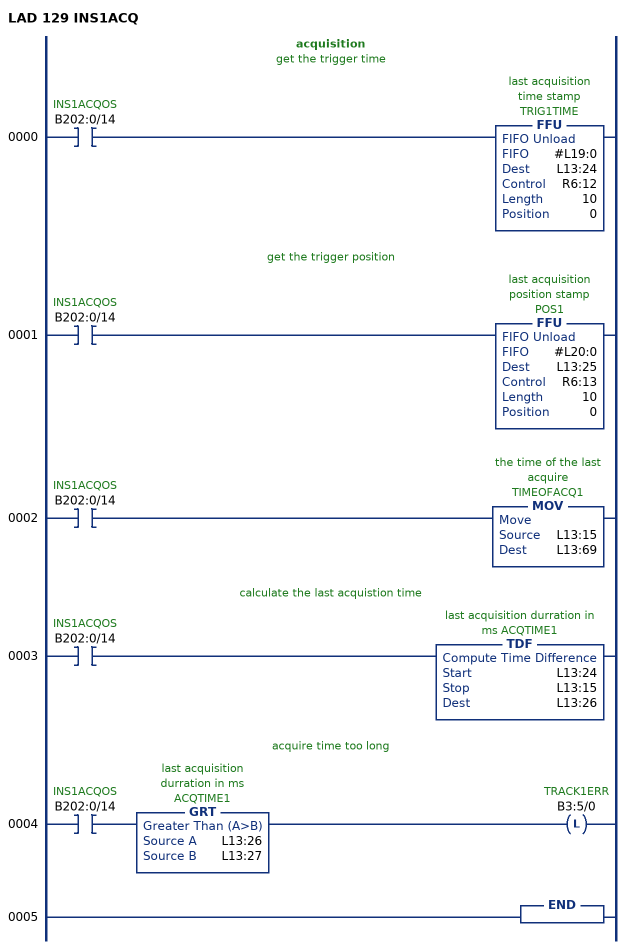
% Rung: 0 %
% TITLE: acquisition %
% get the trigger time %
SOR XIC B202:0/14 FFU #L19:0 L13:24 R6:12 10 0 EOR
%   B202:0/14  INS1ACQOS %
%   L13:24  TRIG1TIME  "last acquisition time stamp" %
% Rung: 1 %
% get the trigger position %
SOR XIC B202:0/14 FFU #L20:0 L13:25 R6:13 10 0 EOR
%   B202:0/14  INS1ACQOS %
%   L13:25  POS1  "last acquisition position stamp" %
% Rung: 2 %
SOR XIC B202:0/14 MOV L13:15 L13:69 EOR
%   B202:0/14  INS1ACQOS %
%   L13:15  THE_TIME %
%   L13:69  TIMEOFACQ1  "the time of the last acquire" %
% Rung: 3 %
% calculate the last acquistion time %
SOR XIC B202:0/14 TDF L13:24 L13:15 L13:26 EOR
%   B202:0/14  INS1ACQOS %
%   L13:24  TRIG1TIME  "last acquisition time stamp" %
%   L13:15  THE_TIME %
%   L13:26  ACQTIME1  "last acquisition durration in ms" %
% Rung: 4 %
% acquire time too long %
SOR XIC B202:0/14 GRT L13:26 L13:27 OTL B3:5/0 EOR
%   B202:0/14  INS1ACQOS %
%   L13:26  ACQTIME1  "last acquisition durration in ms" %
%   L13:27  "max acquisition time in ms" %
%   B3:5/0  TRACK1ERR %
% Rung: 5 %
SOR END EOR

LADDER 130 "INS1TRIG"
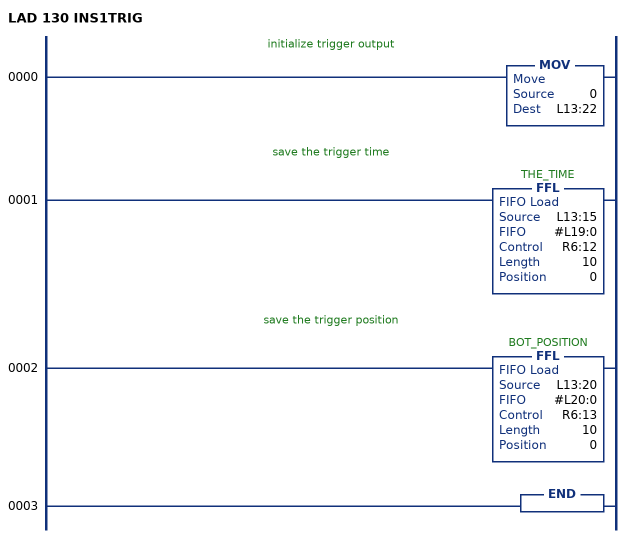
% Rung: 0 %
% initialize trigger output %
SOR MOV 0 L13:22 EOR
% Rung: 1 %
% save the trigger time %
SOR FFL L13:15 #L19:0 R6:12 10 0 EOR
%   L13:15  THE_TIME %
% Rung: 2 %
% save the trigger position %
SOR FFL L13:20 #L20:0 R6:13 10 0 EOR
%   L13:20  BOT_POSITION %
% Rung: 3 %
SOR END EOR

LADDER 131 "XFER"
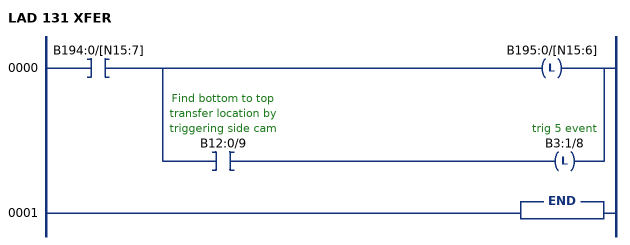
% Rung: 0 %
SOR XIC B194:0/[N15:7] BST OTL B195:0/[N15:6] NXB XIC B12:0/9 OTL B3:1/8 BND EOR
%   N15:7  XFER_OUT_LOC %
%   N15:6  XFER_IN_LOC %
%   B12:0/9  "Find bottom to top transfer location by triggering side cam" %
%   B3:1/8  "trig 5 event" %
% Rung: 1 %
SOR END EOR

LADDER 141 "OPTICTOP"
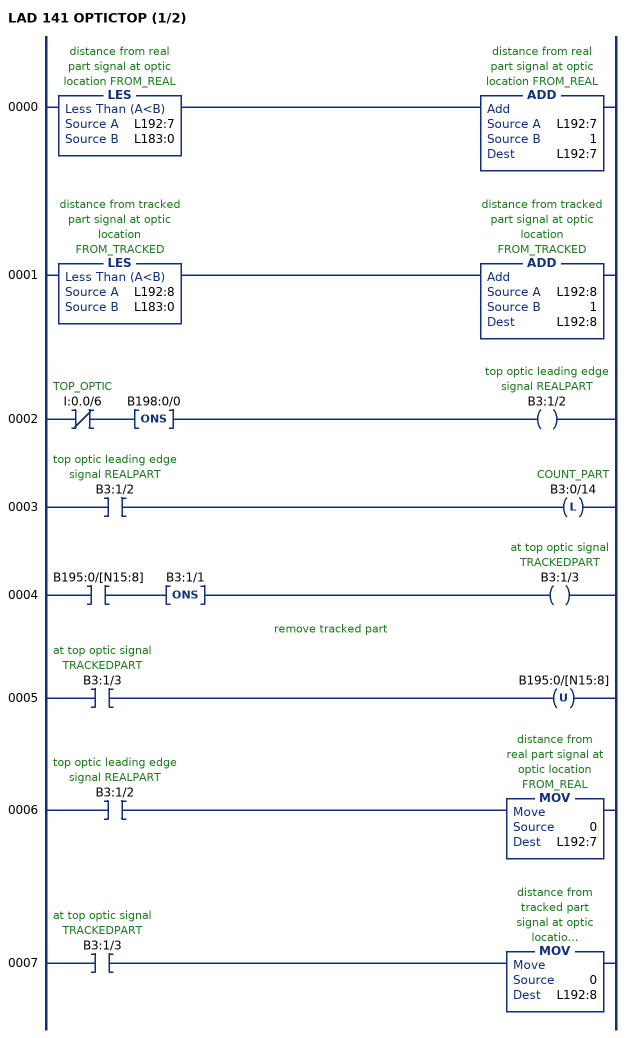
% Rung: 0 %
SOR LES L192:7 L183:0 ADD L192:7 1 L192:7 EOR
%   L192:7  FROM_REAL  "distance from real part signal at optic location" %
% Rung: 1 %
SOR LES L192:8 L183:0 ADD L192:8 1 L192:8 EOR
%   L192:8  FROM_TRACKED  "distance from tracked part signal at optic location" %
% Rung: 2 %
SOR XIO I:0.0/6 ONS B198:0/0 OTE B3:1/2 EOR
%   I:0.0/6  TOP_OPTIC %
%   B3:1/2  REALPART  "top optic leading edge signal" %
% Rung: 3 %
SOR XIC B3:1/2 OTL B3:0/14 EOR
%   B3:1/2  REALPART  "top optic leading edge signal" %
%   B3:0/14  COUNT_PART %
% Rung: 4 %
SOR XIC B195:0/[N15:8] ONS B3:1/1 OTE B3:1/3 EOR
%   N15:8  TOP_OPTIC_LOC %
%   B3:1/3  TRACKEDPART  "at top optic signal" %
% Rung: 5 %
% remove tracked part %
SOR XIC B3:1/3 OTU B195:0/[N15:8] EOR
%   B3:1/3  TRACKEDPART  "at top optic signal" %
%   N15:8  TOP_OPTIC_LOC %
% Rung: 6 %
SOR XIC B3:1/2 MOV 0 L192:7 EOR
%   B3:1/2  REALPART  "top optic leading edge signal" %
%   L192:7  FROM_REAL  "distance from real part signal at optic location" %
% Rung: 7 %
SOR XIC B3:1/3 MOV 0 L192:8 EOR
%   B3:1/3  TRACKEDPART  "at top optic signal" %
%   L192:8  FROM_TRACKED  "distance from tracked part signal at optic location" %

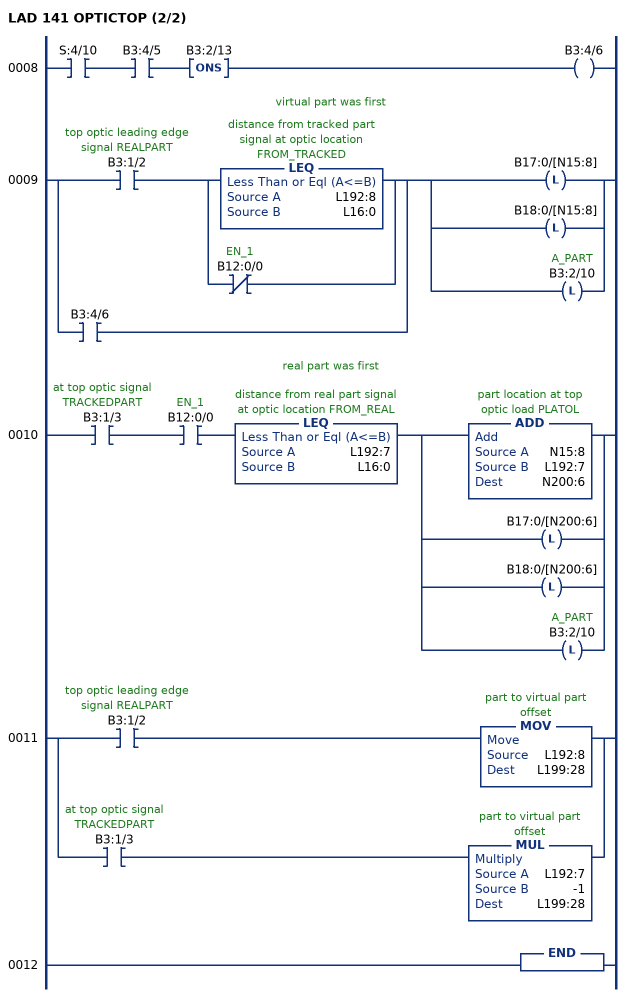
% Rung: 8 %
SOR XIC S:4/10 XIC B3:4/5 ONS B3:2/13 OTE B3:4/6 EOR
% Rung: 9 %
% virtual part was first %
SOR BST XIC B3:1/2 BST LEQ L192:8 L16:0 NXB XIO B12:0/0 BND NXB XIC B3:4/6 BND BST OTL B17:0/[N15:8] NXB OTL B18:0/[N15:8] NXB OTL B3:2/10 BND EOR
%   B3:1/2  REALPART  "top optic leading edge signal" %
%   L192:8  FROM_TRACKED  "distance from tracked part signal at optic location" %
%   B12:0/0  EN_1 %
%   N15:8  TOP_OPTIC_LOC %
%   B3:2/10  A_PART %
% Rung: 10 %
% real part was first %
SOR XIC B3:1/3 XIC B12:0/0 LEQ L192:7 L16:0 BST ADD N15:8 L192:7 N200:6 NXB OTL B17:0/[N200:6] NXB OTL B18:0/[N200:6] NXB OTL B3:2/10 BND EOR
%   B3:1/3  TRACKEDPART  "at top optic signal" %
%   B12:0/0  EN_1 %
%   L192:7  FROM_REAL  "distance from real part signal at optic location" %
%   N15:8  TOP_OPTIC_LOC %
%   N200:6  PLATOL  "part location at top optic load" %
%   B3:2/10  A_PART %
% Rung: 11 %
SOR BST XIC B3:1/2 MOV L192:8 L199:28 NXB XIC B3:1/3 MUL L192:7 -1 L199:28 BND EOR
%   B3:1/2  REALPART  "top optic leading edge signal" %
%   L192:8  FROM_TRACKED  "distance from tracked part signal at optic location" %
%   L199:28  "part to virtual part offset" %
%   B3:1/3  TRACKEDPART  "at top optic signal" %
%   L192:7  FROM_REAL  "distance from real part signal at optic location" %
% Rung: 12 %
SOR END EOR

LADDER 150 "INS 5 MOVE"
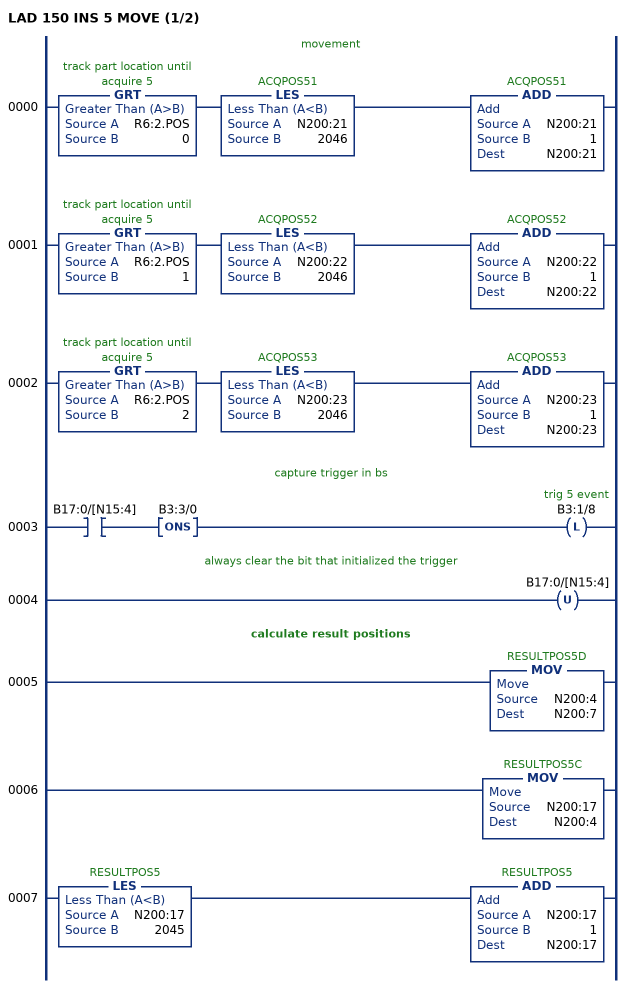
% Rung: 0 %
% movement %
SOR GRT R6:2.POS 0 LES N200:21 2046 ADD N200:21 1 N200:21 EOR
%   R6:2  "track part location until acquire 5" %
%   N200:21  ACQPOS51 %
% Rung: 1 %
SOR GRT R6:2.POS 1 LES N200:22 2046 ADD N200:22 1 N200:22 EOR
%   R6:2  "track part location until acquire 5" %
%   N200:22  ACQPOS52 %
% Rung: 2 %
SOR GRT R6:2.POS 2 LES N200:23 2046 ADD N200:23 1 N200:23 EOR
%   R6:2  "track part location until acquire 5" %
%   N200:23  ACQPOS53 %
% Rung: 3 %
% capture trigger in bs %
SOR XIC B17:0/[N15:4] ONS B3:3/0 OTL B3:1/8 EOR
%   N15:4  INS_5_TRIG_LOC %
%   B3:1/8  "trig 5 event" %
% Rung: 4 %
% always clear the bit that initialized the trigger %
SOR OTU B17:0/[N15:4] EOR
%   N15:4  INS_5_TRIG_LOC %
% Rung: 5 %
% TITLE: calculate result positions %
SOR MOV N200:4 N200:7 EOR
%   N200:4  RESULTPOS5C %
%   N200:7  RESULTPOS5D %
% Rung: 6 %
SOR MOV N200:17 N200:4 EOR
%   N200:17  RESULTPOS5 %
%   N200:4  RESULTPOS5C %
% Rung: 7 %
SOR LES N200:17 2045 ADD N200:17 1 N200:17 EOR
%   N200:17  RESULTPOS5 %

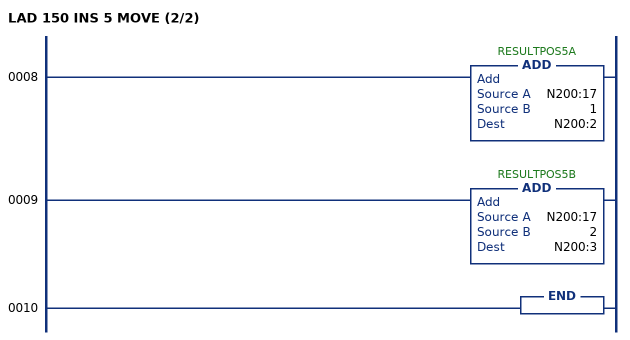
% Rung: 8 %
SOR ADD N200:17 1 N200:2 EOR
%   N200:17  RESULTPOS5 %
%   N200:2  RESULTPOS5A %
% Rung: 9 %
SOR ADD N200:17 2 N200:3 EOR
%   N200:17  RESULTPOS5 %
%   N200:3  RESULTPOS5B %
% Rung: 10 %
SOR END EOR

LADDER 151 "INS 6 MOVE"
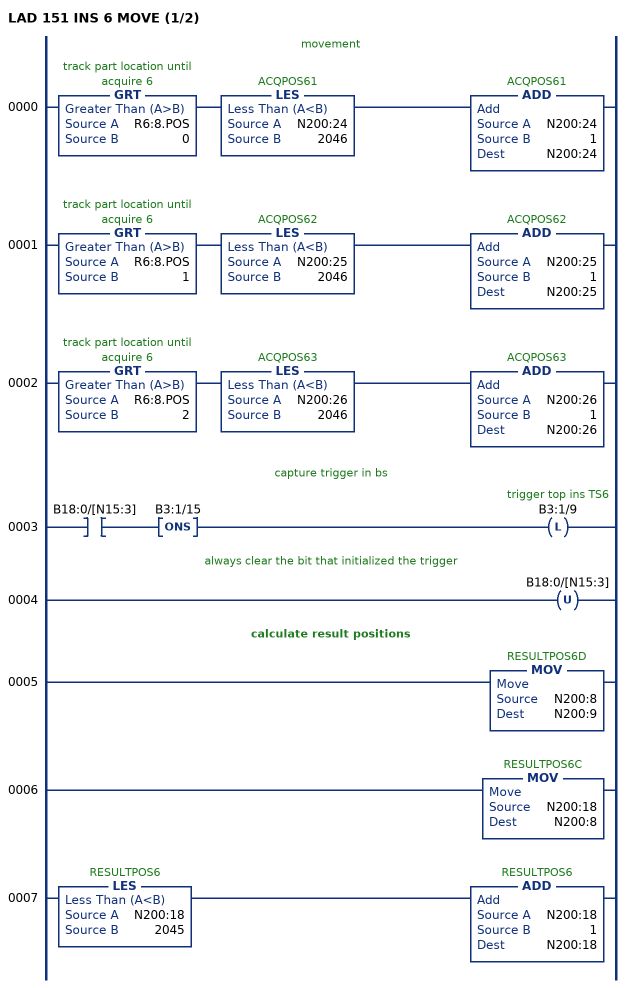
% Rung: 0 %
% movement %
SOR GRT R6:8.POS 0 LES N200:24 2046 ADD N200:24 1 N200:24 EOR
%   R6:8  "track part location until acquire 6" %
%   N200:24  ACQPOS61 %
% Rung: 1 %
SOR GRT R6:8.POS 1 LES N200:25 2046 ADD N200:25 1 N200:25 EOR
%   R6:8  "track part location until acquire 6" %
%   N200:25  ACQPOS62 %
% Rung: 2 %
SOR GRT R6:8.POS 2 LES N200:26 2046 ADD N200:26 1 N200:26 EOR
%   R6:8  "track part location until acquire 6" %
%   N200:26  ACQPOS63 %
% Rung: 3 %
% capture trigger in bs %
SOR XIC B18:0/[N15:3] ONS B3:1/15 OTL B3:1/9 EOR
%   N15:3  INS_6_TRIG_LOC %
%   B3:1/9  TS6  "trigger top ins" %
% Rung: 4 %
% always clear the bit that initialized the trigger %
SOR OTU B18:0/[N15:3] EOR
%   N15:3  INS_6_TRIG_LOC %
% Rung: 5 %
% TITLE: calculate result positions %
SOR MOV N200:8 N200:9 EOR
%   N200:8  RESULTPOS6C %
%   N200:9  RESULTPOS6D %
% Rung: 6 %
SOR MOV N200:18 N200:8 EOR
%   N200:18  RESULTPOS6 %
%   N200:8  RESULTPOS6C %
% Rung: 7 %
SOR LES N200:18 2045 ADD N200:18 1 N200:18 EOR
%   N200:18  RESULTPOS6 %

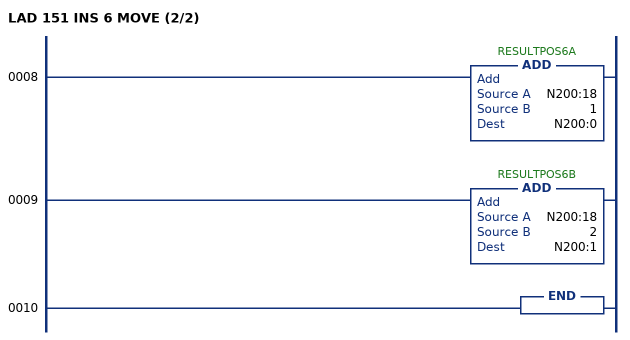
% Rung: 8 %
SOR ADD N200:18 1 N200:0 EOR
%   N200:18  RESULTPOS6 %
%   N200:0  RESULTPOS6A %
% Rung: 9 %
SOR ADD N200:18 2 N200:1 EOR
%   N200:18  RESULTPOS6 %
%   N200:1  RESULTPOS6B %
% Rung: 10 %
SOR END EOR

LADDER 152 "INS 5 NEW"
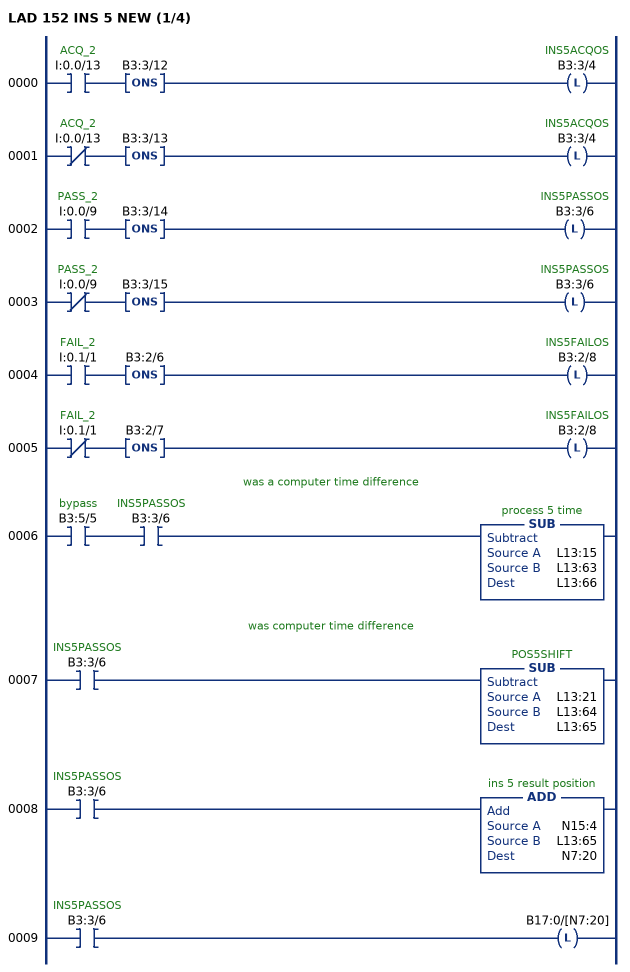
% Rung: 0 %
SOR XIC I:0.0/13 ONS B3:3/12 OTL B3:3/4 EOR
%   I:0.0/13  ACQ_2 %
%   B3:3/4  INS5ACQOS %
% Rung: 1 %
SOR XIO I:0.0/13 ONS B3:3/13 OTL B3:3/4 EOR
%   I:0.0/13  ACQ_2 %
%   B3:3/4  INS5ACQOS %
% Rung: 2 %
SOR XIC I:0.0/9 ONS B3:3/14 OTL B3:3/6 EOR
%   I:0.0/9  PASS_2 %
%   B3:3/6  INS5PASSOS %
% Rung: 3 %
SOR XIO I:0.0/9 ONS B3:3/15 OTL B3:3/6 EOR
%   I:0.0/9  PASS_2 %
%   B3:3/6  INS5PASSOS %
% Rung: 4 %
SOR XIC I:0.1/1 ONS B3:2/6 OTL B3:2/8 EOR
%   I:0.1/1  FAIL_2 %
%   B3:2/8  INS5FAILOS %
% Rung: 5 %
SOR XIO I:0.1/1 ONS B3:2/7 OTL B3:2/8 EOR
%   I:0.1/1  FAIL_2 %
%   B3:2/8  INS5FAILOS %
% Rung: 6 %
% was a computer time difference %
SOR XIC B3:5/5 XIC B3:3/6 SUB L13:15 L13:63 L13:66 EOR
%   B3:5/5  "bypass" %
%   B3:3/6  INS5PASSOS %
%   L13:15  THE_TIME %
%   L13:63  TRIG5TIME  "last acquisition time stamp" %
%   L13:66  "process 5 time" %
% Rung: 7 %
% was computer time difference %
SOR XIC B3:3/6 SUB L13:21 L13:64 L13:65 EOR
%   B3:3/6  INS5PASSOS %
%   L13:21  TOP_POSITION %
%   L13:64  POS5  "last acquisition position stamp" %
%   L13:65  POS5SHIFT %
% Rung: 8 %
SOR XIC B3:3/6 ADD N15:4 L13:65 N7:20 EOR
%   B3:3/6  INS5PASSOS %
%   N15:4  INS_5_TRIG_LOC %
%   L13:65  POS5SHIFT %
%   N7:20  "ins 5 result position" %
% Rung: 9 %
SOR XIC B3:3/6 OTL B17:0/[N7:20] EOR
%   B3:3/6  INS5PASSOS %
%   N7:20  "ins 5 result position" %

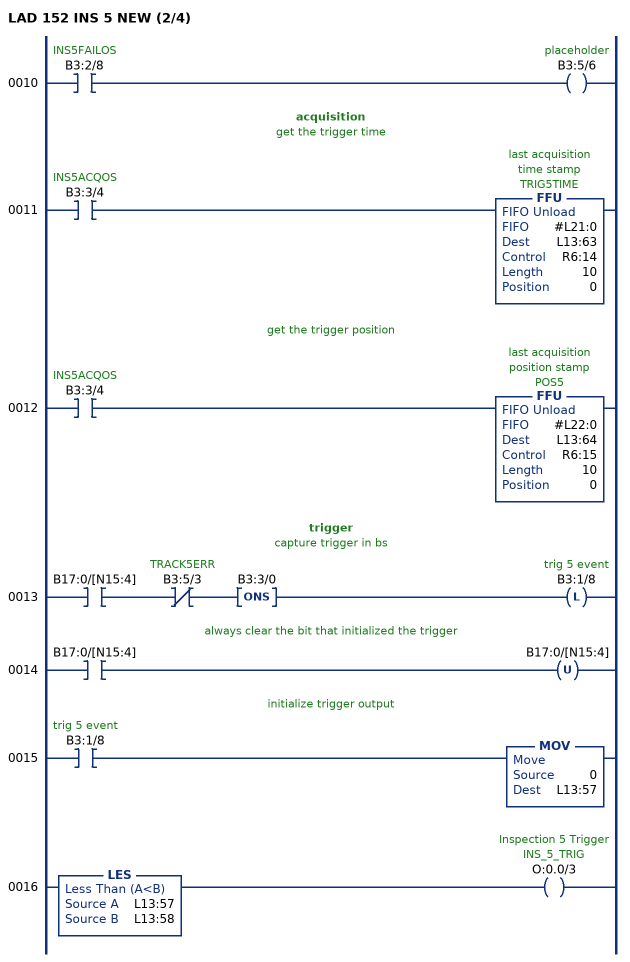
% Rung: 10 %
SOR XIC B3:2/8 OTE B3:5/6 EOR
%   B3:2/8  INS5FAILOS %
%   B3:5/6  "placeholder" %
% Rung: 11 %
% TITLE: acquisition %
% get the trigger time %
SOR XIC B3:3/4 FFU #L21:0 L13:63 R6:14 10 0 EOR
%   B3:3/4  INS5ACQOS %
%   L13:63  TRIG5TIME  "last acquisition time stamp" %
% Rung: 12 %
% get the trigger position %
SOR XIC B3:3/4 FFU #L22:0 L13:64 R6:15 10 0 EOR
%   B3:3/4  INS5ACQOS %
%   L13:64  POS5  "last acquisition position stamp" %
% Rung: 13 %
% TITLE: trigger %
% capture trigger in bs %
SOR XIC B17:0/[N15:4] XIO B3:5/3 ONS B3:3/0 OTL B3:1/8 EOR
%   N15:4  INS_5_TRIG_LOC %
%   B3:5/3  TRACK5ERR %
%   B3:1/8  "trig 5 event" %
% Rung: 14 %
% always clear the bit that initialized the trigger %
SOR XIC B17:0/[N15:4] OTU B17:0/[N15:4] EOR
%   N15:4  INS_5_TRIG_LOC %
% Rung: 15 %
% initialize trigger output %
SOR XIC B3:1/8 MOV 0 L13:57 EOR
%   B3:1/8  "trig 5 event" %
% Rung: 16 %
SOR LES L13:57 L13:58 OTE O:0.0/3 EOR
%   O:0.0/3  INS_5_TRIG  "Inspection 5 Trigger" %

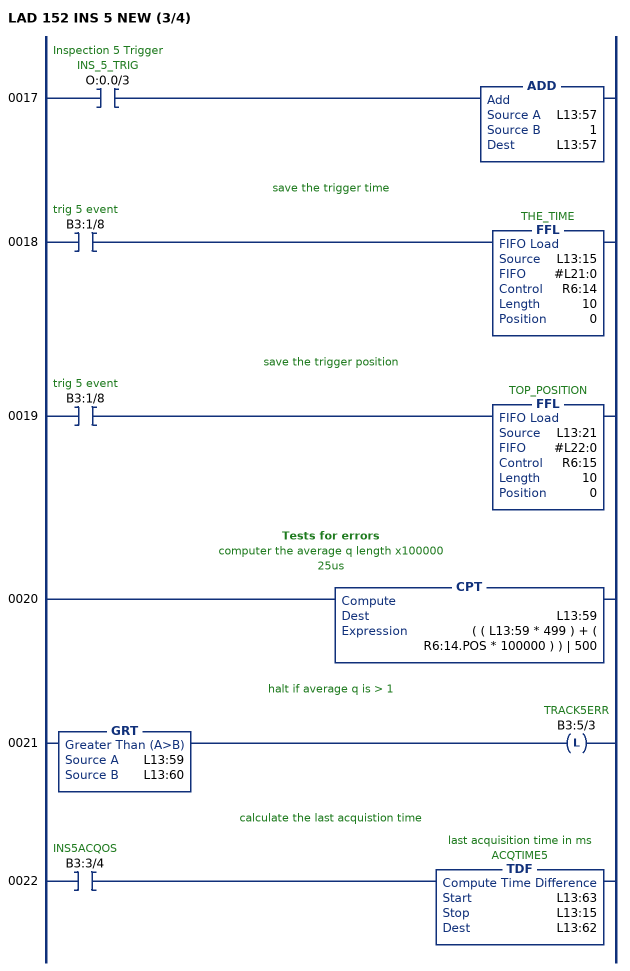
% Rung: 17 %
SOR XIC O:0.0/3 ADD L13:57 1 L13:57 EOR
%   O:0.0/3  INS_5_TRIG  "Inspection 5 Trigger" %
% Rung: 18 %
% save the trigger time %
SOR XIC B3:1/8 FFL L13:15 #L21:0 R6:14 10 0 EOR
%   B3:1/8  "trig 5 event" %
%   L13:15  THE_TIME %
% Rung: 19 %
% save the trigger position %
SOR XIC B3:1/8 FFL L13:21 #L22:0 R6:15 10 0 EOR
%   B3:1/8  "trig 5 event" %
%   L13:21  TOP_POSITION %
% Rung: 20 %
% TITLE: Tests for errors %
% computer the average q length x100000
% 25us %
SOR CPT L13:59 " ( ( L13:59 * 499 ) + ( R6:14.POS * 100000 ) ) | 500 " EOR
% Rung: 21 %
% halt if average q is > 1 %
SOR GRT L13:59 L13:60 OTL B3:5/3 EOR
%   B3:5/3  TRACK5ERR %
% Rung: 22 %
% calculate the last acquistion time %
SOR XIC B3:3/4 TDF L13:63 L13:15 L13:62 EOR
%   B3:3/4  INS5ACQOS %
%   L13:63  TRIG5TIME  "last acquisition time stamp" %
%   L13:15  THE_TIME %
%   L13:62  ACQTIME5  "last acquisition time in ms" %

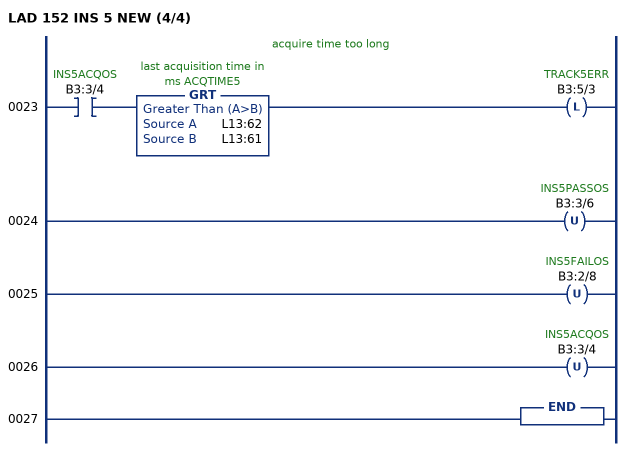
% Rung: 23 %
% acquire time too long %
SOR XIC B3:3/4 GRT L13:62 L13:61 OTL B3:5/3 EOR
%   B3:3/4  INS5ACQOS %
%   L13:62  ACQTIME5  "last acquisition time in ms" %
%   L13:61  "max acquisition time in ms" %
%   B3:5/3  TRACK5ERR %
% Rung: 24 %
SOR OTU B3:3/6 EOR
%   B3:3/6  INS5PASSOS %
% Rung: 25 %
SOR OTU B3:2/8 EOR
%   B3:2/8  INS5FAILOS %
% Rung: 26 %
SOR OTU B3:3/4 EOR
%   B3:3/4  INS5ACQOS %
% Rung: 27 %
SOR END EOR

LADDER 160 "INS 5 TIME"
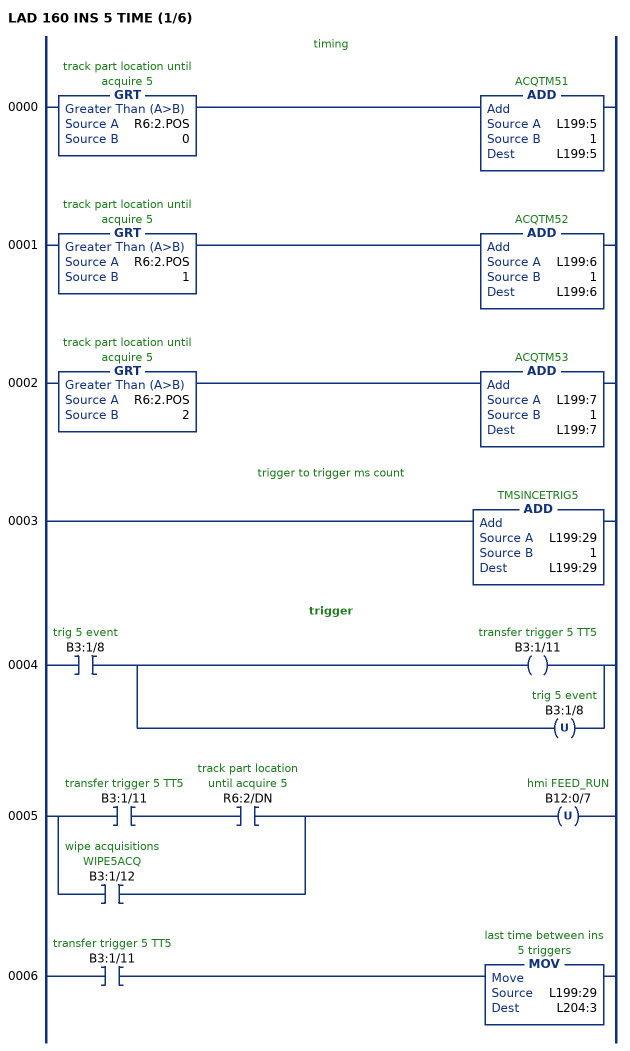
% Rung: 0 %
% timing %
SOR GRT R6:2.POS 0 ADD L199:5 1 L199:5 EOR
%   R6:2  "track part location until acquire 5" %
%   L199:5  ACQTM51 %
% Rung: 1 %
SOR GRT R6:2.POS 1 ADD L199:6 1 L199:6 EOR
%   R6:2  "track part location until acquire 5" %
%   L199:6  ACQTM52 %
% Rung: 2 %
SOR GRT R6:2.POS 2 ADD L199:7 1 L199:7 EOR
%   R6:2  "track part location until acquire 5" %
%   L199:7  ACQTM53 %
% Rung: 3 %
% trigger to trigger ms count %
SOR ADD L199:29 1 L199:29 EOR
%   L199:29  TMSINCETRIG5 %
% Rung: 4 %
% TITLE: trigger %
SOR XIC B3:1/8 BST OTE B3:1/11 NXB OTU B3:1/8 BND EOR
%   B3:1/8  "trig 5 event" %
%   B3:1/11  TT5  "transfer trigger 5" %
% Rung: 5 %
SOR BST XIC B3:1/11 XIC R6:2/DN NXB XIC B3:1/12 BND OTU B12:0/7 EOR
%   B3:1/11  TT5  "transfer trigger 5" %
%   R6:2  "track part location until acquire 5" %
%   B3:1/12  WIPE5ACQ  "wipe acquisitions" %
%   B12:0/7  FEED_RUN  "hmi" %
% Rung: 6 %
SOR XIC B3:1/11 MOV L199:29 L204:3 EOR
%   B3:1/11  TT5  "transfer trigger 5" %
%   L199:29  TMSINCETRIG5 %
%   L204:3  "last time between ins 5 triggers" %

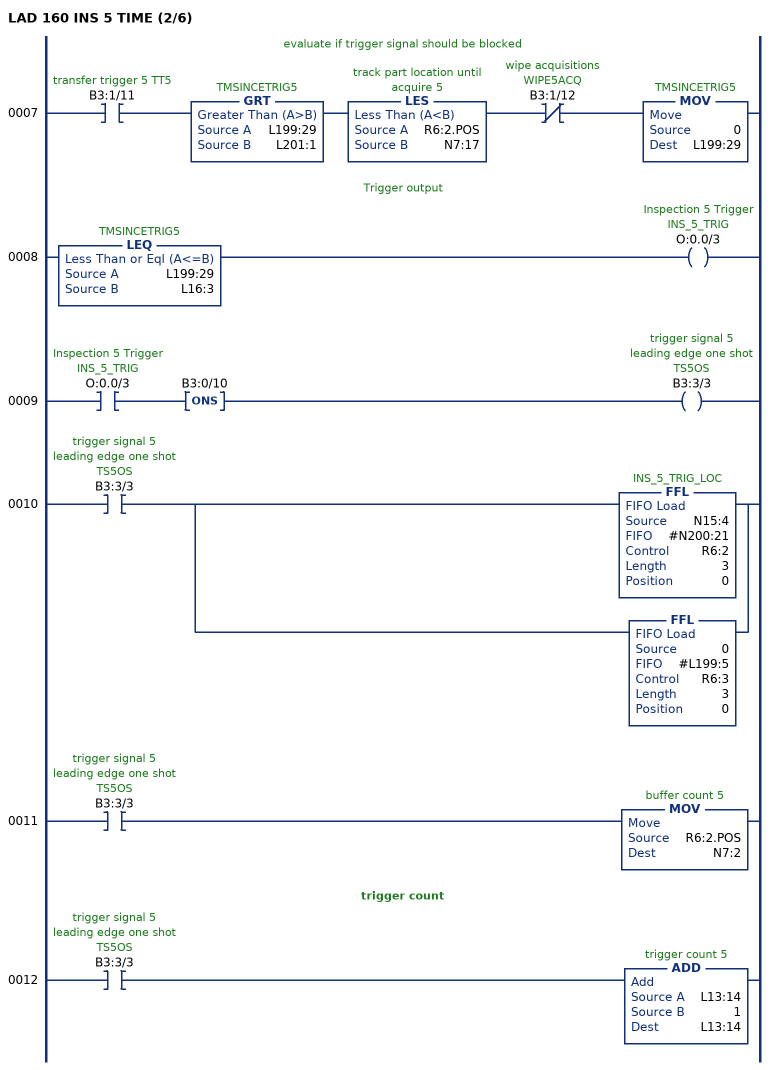
% Rung: 7 %
% evaluate if trigger signal should be blocked %
SOR XIC B3:1/11 GRT L199:29 L201:1 LES R6:2.POS N7:17 XIO B3:1/12 MOV 0 L199:29 EOR
%   B3:1/11  TT5  "transfer trigger 5" %
%   L199:29  TMSINCETRIG5 %
%   L201:1  CAM_5_MIN_CY %
%   R6:2  "track part location until acquire 5" %
%   B3:1/12  WIPE5ACQ  "wipe acquisitions" %
% Rung: 8 %
% Trigger output %
SOR LEQ L199:29 L16:3 OTE O:0.0/3 EOR
%   L199:29  TMSINCETRIG5 %
%   L16:3  CAM_5_TRIG_TIME %
%   O:0.0/3  INS_5_TRIG  "Inspection 5 Trigger" %
% Rung: 9 %
SOR XIC O:0.0/3 ONS B3:0/10 OTE B3:3/3 EOR
%   O:0.0/3  INS_5_TRIG  "Inspection 5 Trigger" %
%   B3:3/3  TS5OS  "trigger signal 5 leading edge one shot" %
% Rung: 10 %
SOR XIC B3:3/3 BST FFL N15:4 #N200:21 R6:2 3 0 NXB FFL 0 #L199:5 R6:3 3 0 BND EOR
%   B3:3/3  TS5OS  "trigger signal 5 leading edge one shot" %
%   N15:4  INS_5_TRIG_LOC %
%   N200:21  ACQPOS51 %
%   R6:2  "track part location until acquire 5" %
%   L199:5  ACQTM51 %
%   R6:3  "track acquire time 5" %
% Rung: 11 %
SOR XIC B3:3/3 MOV R6:2.POS N7:2 EOR
%   B3:3/3  TS5OS  "trigger signal 5 leading edge one shot" %
%   R6:2  "track part location until acquire 5" %
%   N7:2  "buffer count 5" %
% Rung: 12 %
% TITLE: trigger count %
SOR XIC B3:3/3 ADD L13:14 1 L13:14 EOR
%   B3:3/3  TS5OS  "trigger signal 5 leading edge one shot" %
%   L13:14  "trigger count 5" %

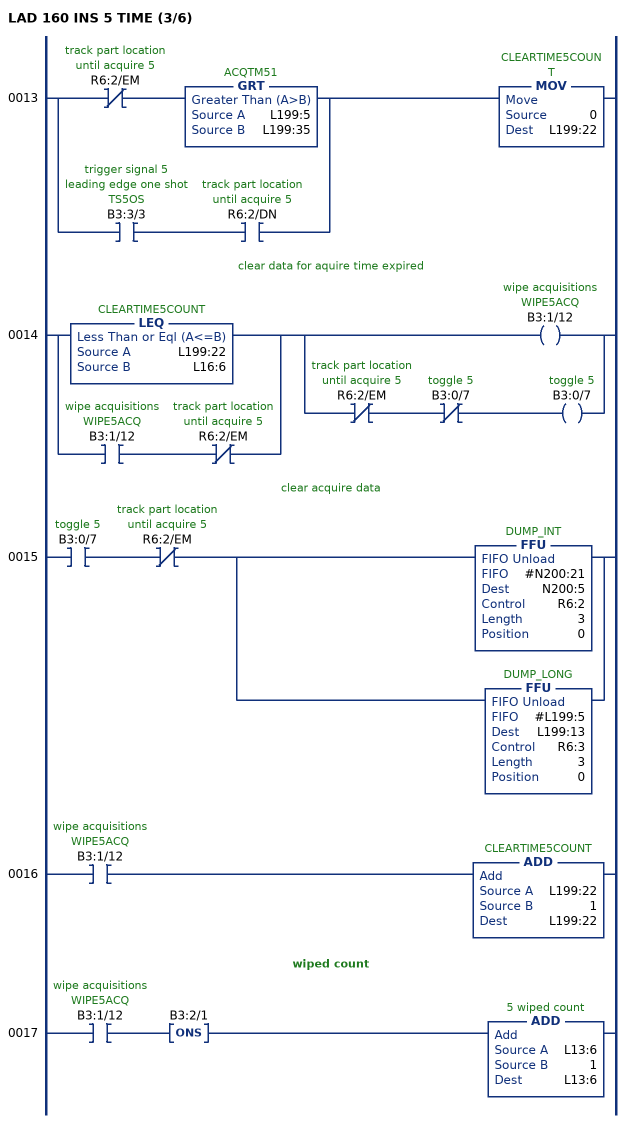
% Rung: 13 %
SOR BST XIO R6:2/EM GRT L199:5 L199:35 NXB XIC B3:3/3 XIC R6:2/DN BND MOV 0 L199:22 EOR
%   R6:2  "track part location until acquire 5" %
%   L199:5  ACQTM51 %
%   L199:35  MAXACQTM5 %
%   B3:3/3  TS5OS  "trigger signal 5 leading edge one shot" %
%   L199:22  CLEARTIME5COUNT %
% Rung: 14 %
% clear data for aquire time expired %
SOR BST LEQ L199:22 L16:6 NXB XIC B3:1/12 XIO R6:2/EM BND BST OTE B3:1/12 NXB XIO R6:2/EM XIO B3:0/7 OTE B3:0/7 BND EOR
%   L199:22  CLEARTIME5COUNT %
%   L16:6  CLEARTIME5 %
%   B3:1/12  WIPE5ACQ  "wipe acquisitions" %
%   R6:2  "track part location until acquire 5" %
%   B3:0/7  "toggle 5" %
% Rung: 15 %
% clear acquire data %
SOR XIC B3:0/7 XIO R6:2/EM BST FFU #N200:21 N200:5 R6:2 3 0 NXB FFU #L199:5 L199:13 R6:3 3 0 BND EOR
%   B3:0/7  "toggle 5" %
%   R6:2  "track part location until acquire 5" %
%   N200:21  ACQPOS51 %
%   N200:5  DUMP_INT %
%   L199:5  ACQTM51 %
%   L199:13  DUMP_LONG %
%   R6:3  "track acquire time 5" %
% Rung: 16 %
SOR XIC B3:1/12 ADD L199:22 1 L199:22 EOR
%   B3:1/12  WIPE5ACQ  "wipe acquisitions" %
%   L199:22  CLEARTIME5COUNT %
% Rung: 17 %
% TITLE: wiped count %
SOR XIC B3:1/12 ONS B3:2/1 ADD L13:6 1 L13:6 EOR
%   B3:1/12  WIPE5ACQ  "wipe acquisitions" %
%   L13:6  "5 wiped count" %

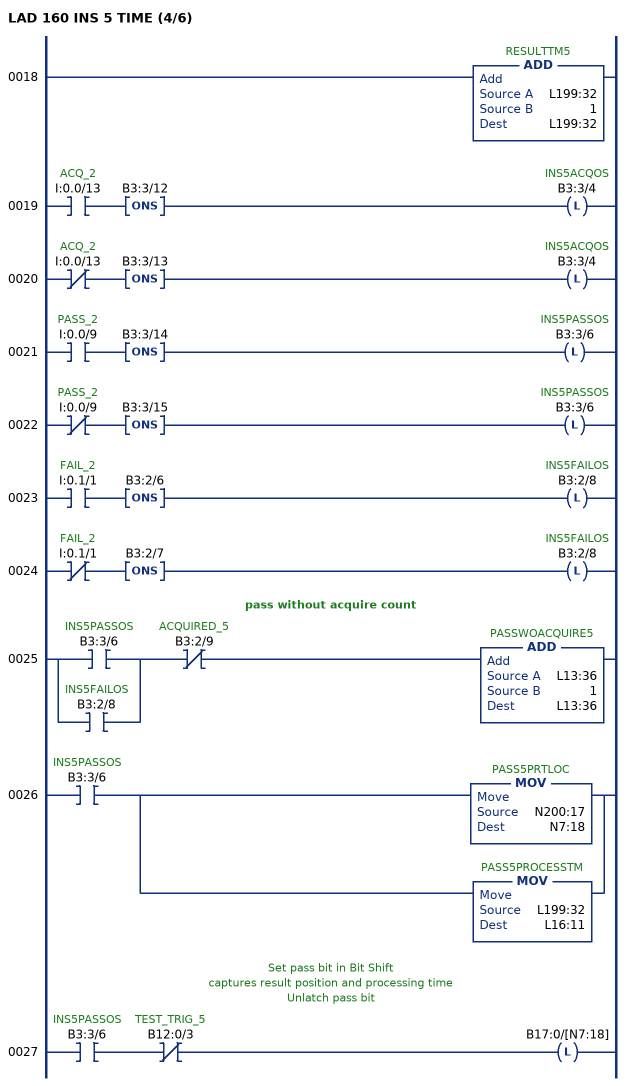
% Rung: 18 %
SOR ADD L199:32 1 L199:32 EOR
%   L199:32  RESULTTM5 %
% Rung: 19 %
SOR XIC I:0.0/13 ONS B3:3/12 OTL B3:3/4 EOR
%   I:0.0/13  ACQ_2 %
%   B3:3/4  INS5ACQOS %
% Rung: 20 %
SOR XIO I:0.0/13 ONS B3:3/13 OTL B3:3/4 EOR
%   I:0.0/13  ACQ_2 %
%   B3:3/4  INS5ACQOS %
% Rung: 21 %
SOR XIC I:0.0/9 ONS B3:3/14 OTL B3:3/6 EOR
%   I:0.0/9  PASS_2 %
%   B3:3/6  INS5PASSOS %
% Rung: 22 %
SOR XIO I:0.0/9 ONS B3:3/15 OTL B3:3/6 EOR
%   I:0.0/9  PASS_2 %
%   B3:3/6  INS5PASSOS %
% Rung: 23 %
SOR XIC I:0.1/1 ONS B3:2/6 OTL B3:2/8 EOR
%   I:0.1/1  FAIL_2 %
%   B3:2/8  INS5FAILOS %
% Rung: 24 %
SOR XIO I:0.1/1 ONS B3:2/7 OTL B3:2/8 EOR
%   I:0.1/1  FAIL_2 %
%   B3:2/8  INS5FAILOS %
% Rung: 25 %
% TITLE: pass without acquire count %
SOR BST XIC B3:3/6 NXB XIC B3:2/8 BND XIO B3:2/9 ADD L13:36 1 L13:36 EOR
%   B3:3/6  INS5PASSOS %
%   B3:2/8  INS5FAILOS %
%   B3:2/9  ACQUIRED_5 %
%   L13:36  PASSWOACQUIRE5 %
% Rung: 26 %
SOR XIC B3:3/6 BST MOV N200:17 N7:18 NXB MOV L199:32 L16:11 BND EOR
%   B3:3/6  INS5PASSOS %
%   N200:17  RESULTPOS5 %
%   N7:18  PASS5PRTLOC %
%   L199:32  RESULTTM5 %
%   L16:11  PASS5PROCESSTM %
% Rung: 27 %
% Set pass bit in Bit Shift
% captures result position and processing time
% Unlatch pass bit %
SOR XIC B3:3/6 XIO B12:0/3 OTL B17:0/[N7:18] EOR
%   B3:3/6  INS5PASSOS %
%   B12:0/3  TEST_TRIG_5 %
%   N7:18  PASS5PRTLOC %

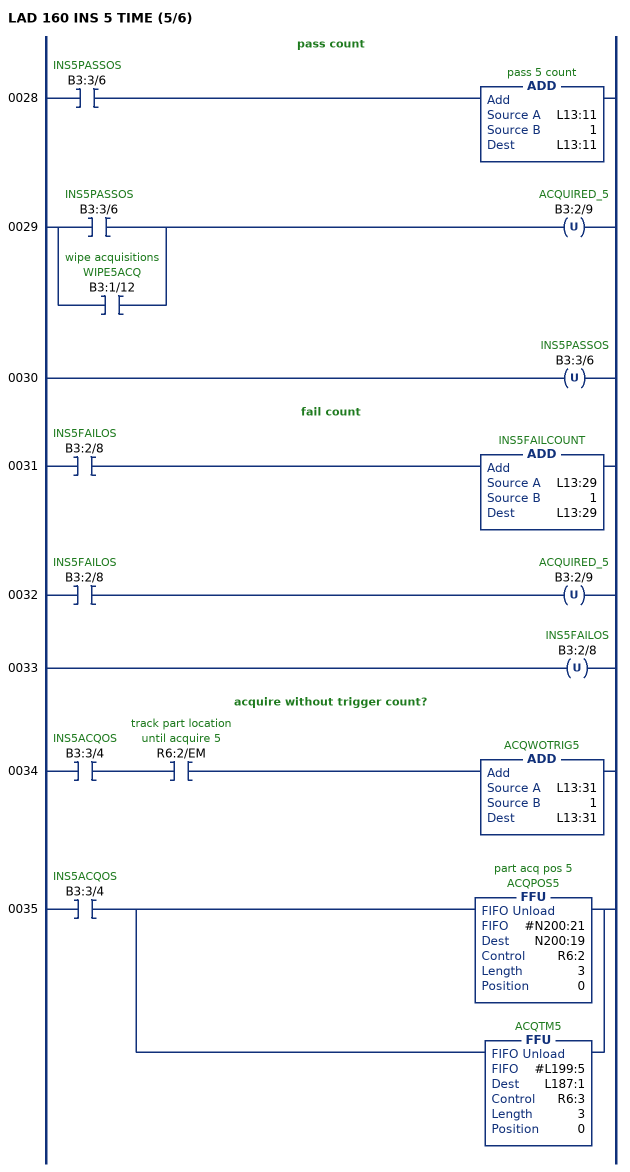
% Rung: 28 %
% TITLE: pass count %
SOR XIC B3:3/6 ADD L13:11 1 L13:11 EOR
%   B3:3/6  INS5PASSOS %
%   L13:11  "pass 5 count" %
% Rung: 29 %
SOR BST XIC B3:3/6 NXB XIC B3:1/12 BND OTU B3:2/9 EOR
%   B3:3/6  INS5PASSOS %
%   B3:1/12  WIPE5ACQ  "wipe acquisitions" %
%   B3:2/9  ACQUIRED_5 %
% Rung: 30 %
SOR OTU B3:3/6 EOR
%   B3:3/6  INS5PASSOS %
% Rung: 31 %
% TITLE: fail count %
SOR XIC B3:2/8 ADD L13:29 1 L13:29 EOR
%   B3:2/8  INS5FAILOS %
%   L13:29  INS5FAILCOUNT %
% Rung: 32 %
SOR XIC B3:2/8 OTU B3:2/9 EOR
%   B3:2/8  INS5FAILOS %
%   B3:2/9  ACQUIRED_5 %
% Rung: 33 %
SOR OTU B3:2/8 EOR
%   B3:2/8  INS5FAILOS %
% Rung: 34 %
% TITLE: acquire without trigger count? %
SOR XIC B3:3/4 XIC R6:2/EM ADD L13:31 1 L13:31 EOR
%   B3:3/4  INS5ACQOS %
%   R6:2  "track part location until acquire 5" %
%   L13:31  ACQWOTRIG5 %
% Rung: 35 %
SOR XIC B3:3/4 BST FFU #N200:21 N200:19 R6:2 3 0 NXB FFU #L199:5 L187:1 R6:3 3 0 BND EOR
%   B3:3/4  INS5ACQOS %
%   N200:21  ACQPOS51 %
%   N200:19  ACQPOS5  "part acq pos 5" %
%   R6:2  "track part location until acquire 5" %
%   L199:5  ACQTM51 %
%   L187:1  ACQTM5 %
%   R6:3  "track acquire time 5" %

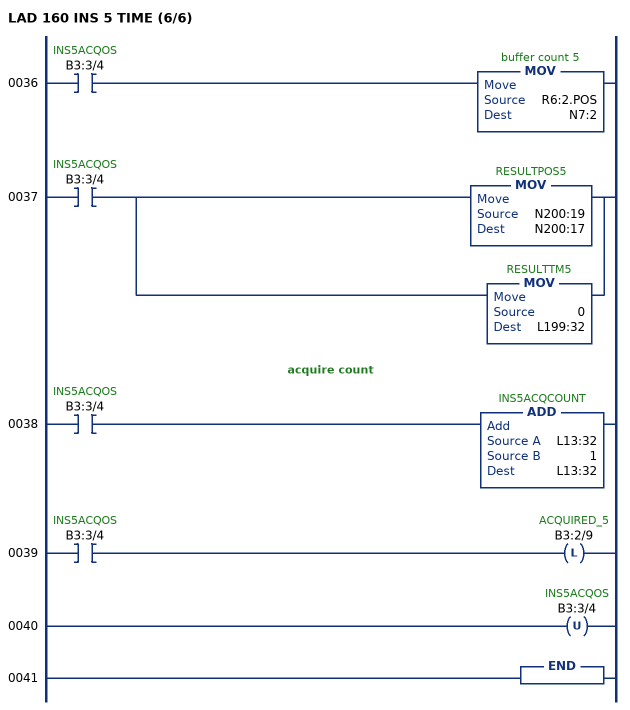
% Rung: 36 %
SOR XIC B3:3/4 MOV R6:2.POS N7:2 EOR
%   B3:3/4  INS5ACQOS %
%   R6:2  "track part location until acquire 5" %
%   N7:2  "buffer count 5" %
% Rung: 37 %
SOR XIC B3:3/4 BST MOV N200:19 N200:17 NXB MOV 0 L199:32 BND EOR
%   B3:3/4  INS5ACQOS %
%   N200:19  ACQPOS5  "part acq pos 5" %
%   N200:17  RESULTPOS5 %
%   L199:32  RESULTTM5 %
% Rung: 38 %
% TITLE: acquire count %
SOR XIC B3:3/4 ADD L13:32 1 L13:32 EOR
%   B3:3/4  INS5ACQOS %
%   L13:32  INS5ACQCOUNT %
% Rung: 39 %
SOR XIC B3:3/4 OTL B3:2/9 EOR
%   B3:3/4  INS5ACQOS %
%   B3:2/9  ACQUIRED_5 %
% Rung: 40 %
SOR OTU B3:3/4 EOR
%   B3:3/4  INS5ACQOS %
% Rung: 41 %
SOR END EOR

LADDER 161 "INS 6 TIME"
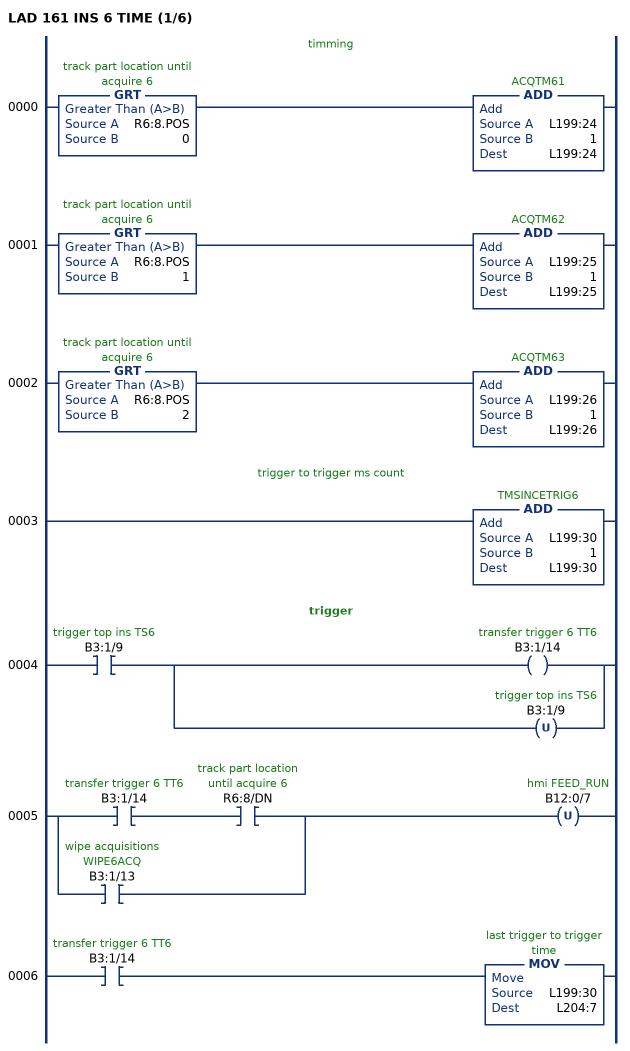
% Rung: 0 %
% timming %
SOR GRT R6:8.POS 0 ADD L199:24 1 L199:24 EOR
%   R6:8  "track part location until acquire 6" %
%   L199:24  ACQTM61 %
% Rung: 1 %
SOR GRT R6:8.POS 1 ADD L199:25 1 L199:25 EOR
%   R6:8  "track part location until acquire 6" %
%   L199:25  ACQTM62 %
% Rung: 2 %
SOR GRT R6:8.POS 2 ADD L199:26 1 L199:26 EOR
%   R6:8  "track part location until acquire 6" %
%   L199:26  ACQTM63 %
% Rung: 3 %
% trigger to trigger ms count %
SOR ADD L199:30 1 L199:30 EOR
%   L199:30  TMSINCETRIG6 %
% Rung: 4 %
% TITLE: trigger %
SOR XIC B3:1/9 BST OTE B3:1/14 NXB OTU B3:1/9 BND EOR
%   B3:1/9  TS6  "trigger top ins" %
%   B3:1/14  TT6  "transfer trigger 6" %
% Rung: 5 %
SOR BST XIC B3:1/14 XIC R6:8/DN NXB XIC B3:1/13 BND OTU B12:0/7 EOR
%   B3:1/14  TT6  "transfer trigger 6" %
%   R6:8  "track part location until acquire 6" %
%   B3:1/13  WIPE6ACQ  "wipe acquisitions" %
%   B12:0/7  FEED_RUN  "hmi" %
% Rung: 6 %
SOR XIC B3:1/14 MOV L199:30 L204:7 EOR
%   B3:1/14  TT6  "transfer trigger 6" %
%   L199:30  TMSINCETRIG6 %
%   L204:7  "last trigger to trigger time" %

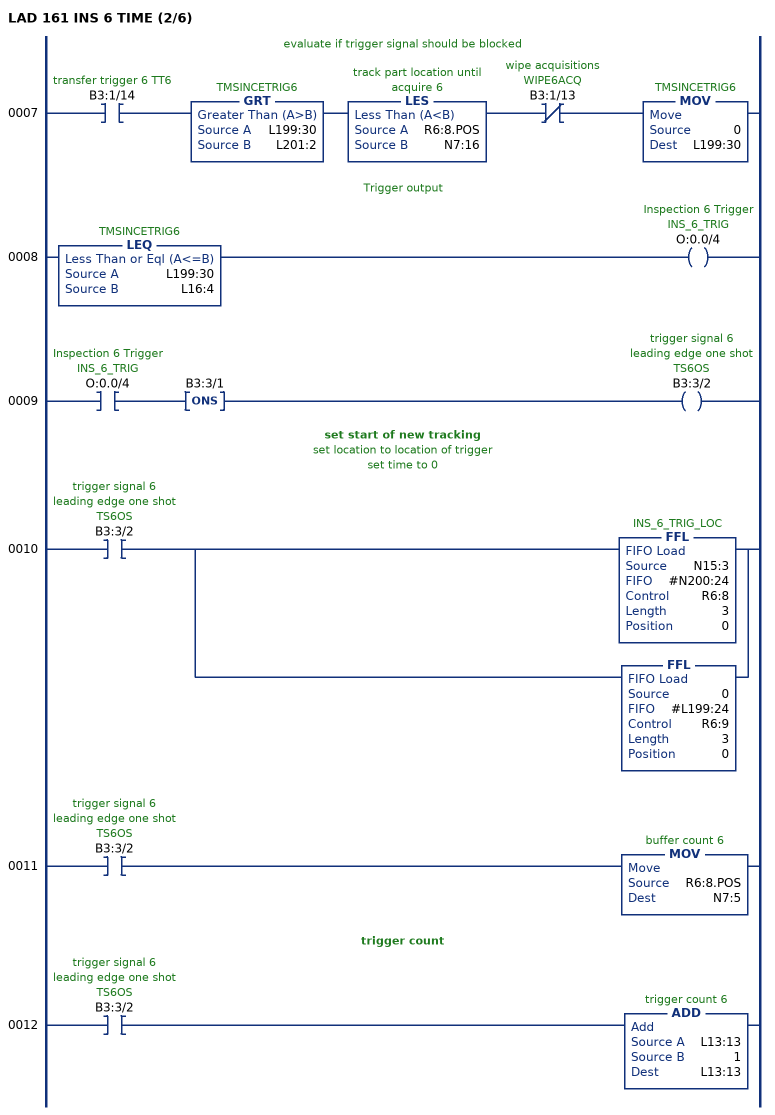
% Rung: 7 %
% evaluate if trigger signal should be blocked %
SOR XIC B3:1/14 GRT L199:30 L201:2 LES R6:8.POS N7:16 XIO B3:1/13 MOV 0 L199:30 EOR
%   B3:1/14  TT6  "transfer trigger 6" %
%   L199:30  TMSINCETRIG6 %
%   L201:2  CAM_6_MIN_CY %
%   R6:8  "track part location until acquire 6" %
%   B3:1/13  WIPE6ACQ  "wipe acquisitions" %
% Rung: 8 %
% Trigger output %
SOR LEQ L199:30 L16:4 OTE O:0.0/4 EOR
%   L199:30  TMSINCETRIG6 %
%   L16:4  CAM_6_TRIG_TIME %
%   O:0.0/4  INS_6_TRIG  "Inspection 6 Trigger" %
% Rung: 9 %
SOR XIC O:0.0/4 ONS B3:3/1 OTE B3:3/2 EOR
%   O:0.0/4  INS_6_TRIG  "Inspection 6 Trigger" %
%   B3:3/2  TS6OS  "trigger signal 6 leading edge one shot" %
% Rung: 10 %
% TITLE: set start of new tracking %
% set location to location of trigger
% set time to 0 %
SOR XIC B3:3/2 BST FFL N15:3 #N200:24 R6:8 3 0 NXB FFL 0 #L199:24 R6:9 3 0 BND EOR
%   B3:3/2  TS6OS  "trigger signal 6 leading edge one shot" %
%   N15:3  INS_6_TRIG_LOC %
%   N200:24  ACQPOS61 %
%   R6:8  "track part location until acquire 6" %
%   L199:24  ACQTM61 %
%   R6:9  "track acquire time 6" %
% Rung: 11 %
SOR XIC B3:3/2 MOV R6:8.POS N7:5 EOR
%   B3:3/2  TS6OS  "trigger signal 6 leading edge one shot" %
%   R6:8  "track part location until acquire 6" %
%   N7:5  "buffer count 6" %
% Rung: 12 %
% TITLE: trigger count %
SOR XIC B3:3/2 ADD L13:13 1 L13:13 EOR
%   B3:3/2  TS6OS  "trigger signal 6 leading edge one shot" %
%   L13:13  "trigger count 6" %

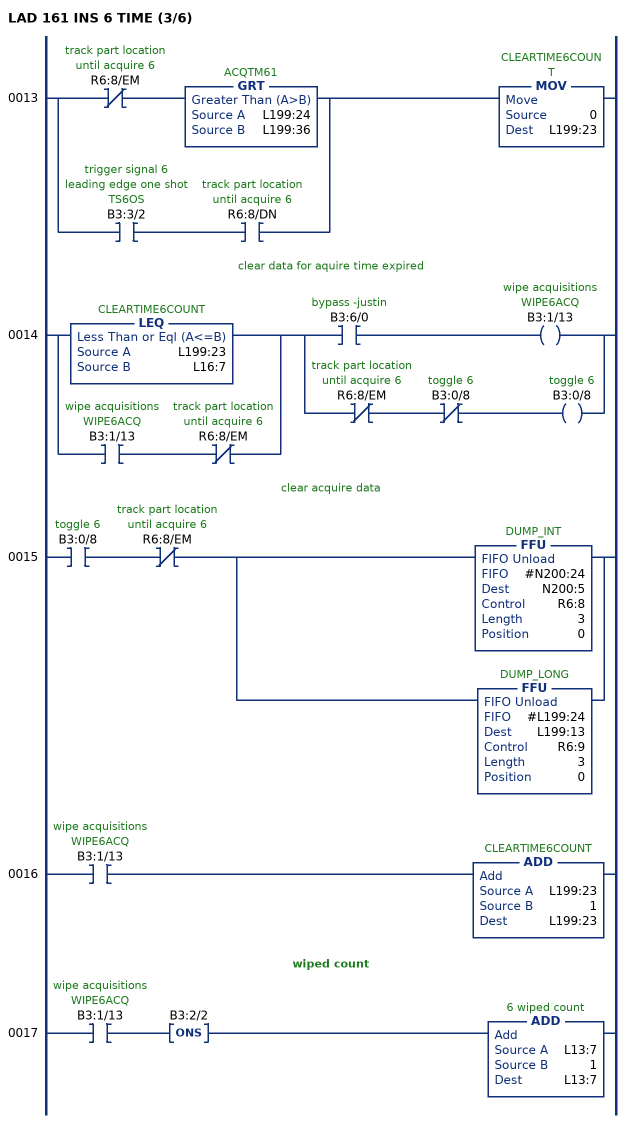
% Rung: 13 %
SOR BST XIO R6:8/EM GRT L199:24 L199:36 NXB XIC B3:3/2 XIC R6:8/DN BND MOV 0 L199:23 EOR
%   R6:8  "track part location until acquire 6" %
%   L199:24  ACQTM61 %
%   L199:36  MAXACQTM6 %
%   B3:3/2  TS6OS  "trigger signal 6 leading edge one shot" %
%   L199:23  CLEARTIME6COUNT %
% Rung: 14 %
% clear data for aquire time expired %
SOR BST LEQ L199:23 L16:7 NXB XIC B3:1/13 XIO R6:8/EM BND BST XIC B3:6/0 OTE B3:1/13 NXB XIO R6:8/EM XIO B3:0/8 OTE B3:0/8 BND EOR
%   L199:23  CLEARTIME6COUNT %
%   L16:7  CLEARTIME6 %
%   B3:1/13  WIPE6ACQ  "wipe acquisitions" %
%   R6:8  "track part location until acquire 6" %
%   B3:6/0  "bypass -justin" %
%   B3:0/8  "toggle 6" %
% Rung: 15 %
% clear acquire data %
SOR XIC B3:0/8 XIO R6:8/EM BST FFU #N200:24 N200:5 R6:8 3 0 NXB FFU #L199:24 L199:13 R6:9 3 0 BND EOR
%   B3:0/8  "toggle 6" %
%   R6:8  "track part location until acquire 6" %
%   N200:24  ACQPOS61 %
%   N200:5  DUMP_INT %
%   L199:24  ACQTM61 %
%   L199:13  DUMP_LONG %
%   R6:9  "track acquire time 6" %
% Rung: 16 %
SOR XIC B3:1/13 ADD L199:23 1 L199:23 EOR
%   B3:1/13  WIPE6ACQ  "wipe acquisitions" %
%   L199:23  CLEARTIME6COUNT %
% Rung: 17 %
% TITLE: wiped count %
SOR XIC B3:1/13 ONS B3:2/2 ADD L13:7 1 L13:7 EOR
%   B3:1/13  WIPE6ACQ  "wipe acquisitions" %
%   L13:7  "6 wiped count" %

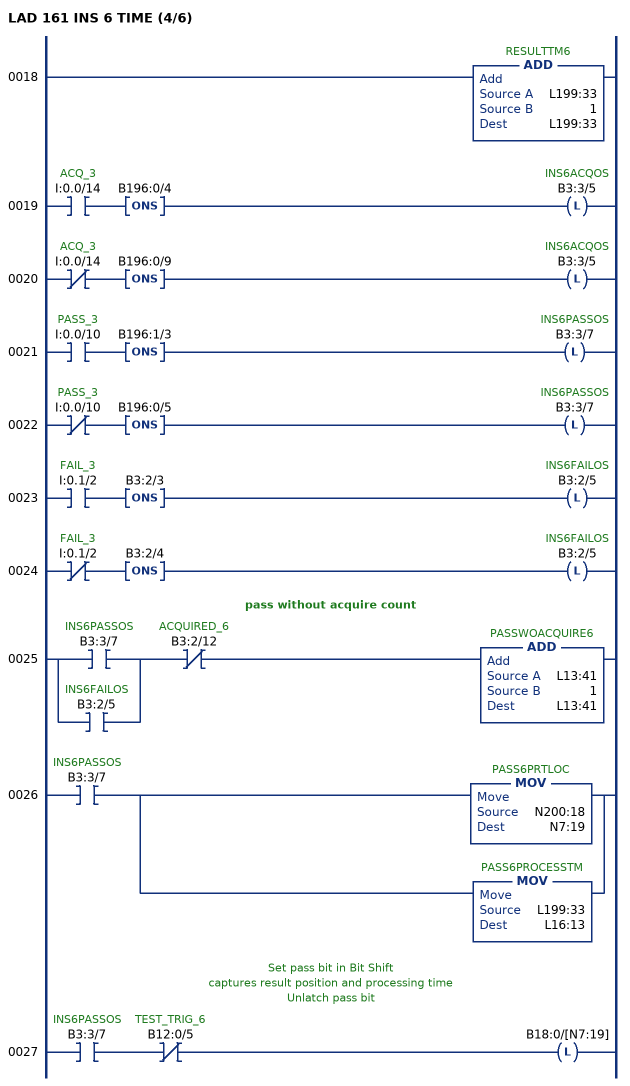
% Rung: 18 %
SOR ADD L199:33 1 L199:33 EOR
%   L199:33  RESULTTM6 %
% Rung: 19 %
SOR XIC I:0.0/14 ONS B196:0/4 OTL B3:3/5 EOR
%   I:0.0/14  ACQ_3 %
%   B3:3/5  INS6ACQOS %
% Rung: 20 %
SOR XIO I:0.0/14 ONS B196:0/9 OTL B3:3/5 EOR
%   I:0.0/14  ACQ_3 %
%   B3:3/5  INS6ACQOS %
% Rung: 21 %
SOR XIC I:0.0/10 ONS B196:1/3 OTL B3:3/7 EOR
%   I:0.0/10  PASS_3 %
%   B3:3/7  INS6PASSOS %
% Rung: 22 %
SOR XIO I:0.0/10 ONS B196:0/5 OTL B3:3/7 EOR
%   I:0.0/10  PASS_3 %
%   B3:3/7  INS6PASSOS %
% Rung: 23 %
SOR XIC I:0.1/2 ONS B3:2/3 OTL B3:2/5 EOR
%   I:0.1/2  FAIL_3 %
%   B3:2/5  INS6FAILOS %
% Rung: 24 %
SOR XIO I:0.1/2 ONS B3:2/4 OTL B3:2/5 EOR
%   I:0.1/2  FAIL_3 %
%   B3:2/5  INS6FAILOS %
% Rung: 25 %
% TITLE: pass without acquire count %
SOR BST XIC B3:3/7 NXB XIC B3:2/5 BND XIO B3:2/12 ADD L13:41 1 L13:41 EOR
%   B3:3/7  INS6PASSOS %
%   B3:2/5  INS6FAILOS %
%   B3:2/12  ACQUIRED_6 %
%   L13:41  PASSWOACQUIRE6 %
% Rung: 26 %
SOR XIC B3:3/7 BST MOV N200:18 N7:19 NXB MOV L199:33 L16:13 BND EOR
%   B3:3/7  INS6PASSOS %
%   N200:18  RESULTPOS6 %
%   N7:19  PASS6PRTLOC %
%   L199:33  RESULTTM6 %
%   L16:13  PASS6PROCESSTM %
% Rung: 27 %
% Set pass bit in Bit Shift
% captures result position and processing time
% Unlatch pass bit %
SOR XIC B3:3/7 XIO B12:0/5 OTL B18:0/[N7:19] EOR
%   B3:3/7  INS6PASSOS %
%   B12:0/5  TEST_TRIG_6 %
%   N7:19  PASS6PRTLOC %

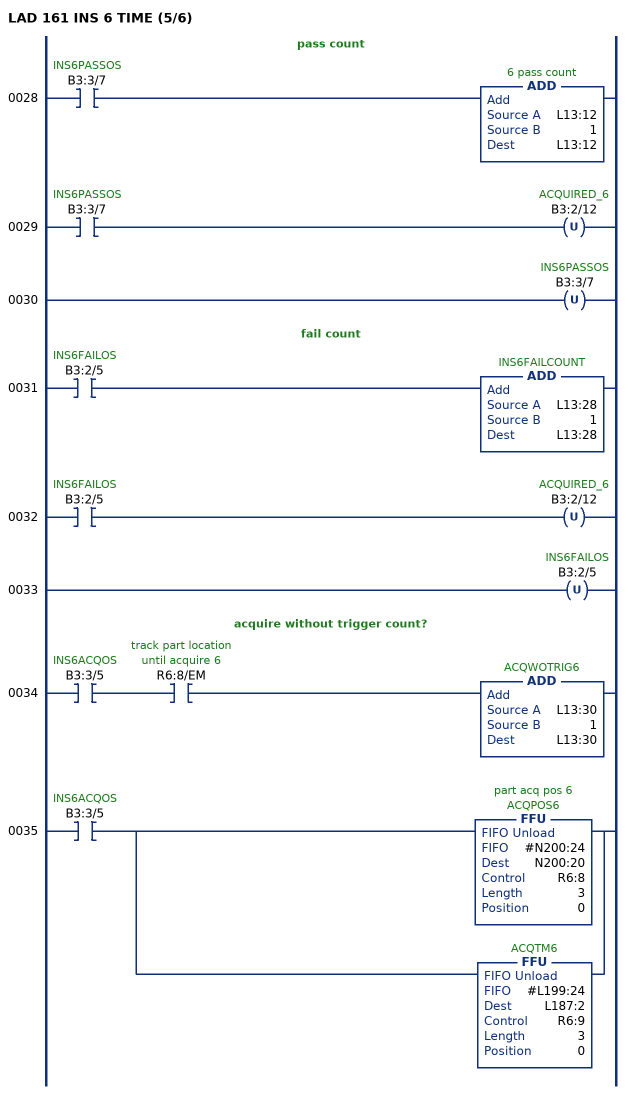
% Rung: 28 %
% TITLE: pass count %
SOR XIC B3:3/7 ADD L13:12 1 L13:12 EOR
%   B3:3/7  INS6PASSOS %
%   L13:12  "6 pass count" %
% Rung: 29 %
SOR XIC B3:3/7 OTU B3:2/12 EOR
%   B3:3/7  INS6PASSOS %
%   B3:2/12  ACQUIRED_6 %
% Rung: 30 %
SOR OTU B3:3/7 EOR
%   B3:3/7  INS6PASSOS %
% Rung: 31 %
% TITLE: fail count %
SOR XIC B3:2/5 ADD L13:28 1 L13:28 EOR
%   B3:2/5  INS6FAILOS %
%   L13:28  INS6FAILCOUNT %
% Rung: 32 %
SOR XIC B3:2/5 OTU B3:2/12 EOR
%   B3:2/5  INS6FAILOS %
%   B3:2/12  ACQUIRED_6 %
% Rung: 33 %
SOR OTU B3:2/5 EOR
%   B3:2/5  INS6FAILOS %
% Rung: 34 %
% TITLE: acquire without trigger count? %
SOR XIC B3:3/5 XIC R6:8/EM ADD L13:30 1 L13:30 EOR
%   B3:3/5  INS6ACQOS %
%   R6:8  "track part location until acquire 6" %
%   L13:30  ACQWOTRIG6 %
% Rung: 35 %
SOR XIC B3:3/5 BST FFU #N200:24 N200:20 R6:8 3 0 NXB FFU #L199:24 L187:2 R6:9 3 0 BND EOR
%   B3:3/5  INS6ACQOS %
%   N200:24  ACQPOS61 %
%   N200:20  ACQPOS6  "part acq pos 6" %
%   R6:8  "track part location until acquire 6" %
%   L199:24  ACQTM61 %
%   L187:2  ACQTM6 %
%   R6:9  "track acquire time 6" %

